// TIA Portal V21 export
TYPE "Std_AllarmiZona"
   STRUCT
      Stato : Bool;   // Stato allarme 0=Non presente 1 = Presente
      Silenziato : Bool;   // Stato tacitazione 0=Non presente 1 = Presente
      Tipo : Byte;   // Classe di caduta ciclo 0=Warning 1=AllarmeAuto 2= AllarmeMan
   END_STRUCT;
END_TYPE
